(* Logix 5000 project; controller cal1632 1756-L62 rev 16.20; software revision 16.05; part 42 of 57 *)
(* tags used below, declared in another part *)
   FAULT : BOOL;
   HMI : BOOL;
   p01r09_pb_global_reset : BOOL;
   p02_real_from_hmi : hmi_real;
   p25_ai_amps : DINT;
   p25_ai_hz : DINT;
   p25_ai_rpm : REAL;
   p25_ai_speed : REAL;
   p25_ai_ts2_lc : REAL;
   p25_ao_selected_speed : REAL;
   p25_ao_torque : REAL;
   p25_ao_vfd : REAL;
   p25_control_word : INT;
   p25_di_brake : BOOL;
   p25_di_therm : BOOL;
   p25_di_ts2 : acs800_di_normal;
   p25_dint_to_hmi : DINT[16];
   p25_real_to_hmi : REAL[112];
   p25_status_word : INT;
   p25_ts2_gear_ratio : REAL;
   p25_ts2_roll_diameter_ft : REAL;
   p25_vfd_input_max : REAL;
   p25_vfd_input_min : REAL;
   p25_vfd_output_max : REAL;
   p25_vfd_output_min : REAL;
   p25r03_vfd_out_scaling : SYS_SCP;
   p25r04 : routine;
   p25r04_speed_to_vfd_ts2_scp : SYS_SPEED_TO_VFD;
   p25r04_timer_fault : TIMER[4];
   p25r04_timer_warning : TIMER[4];
   p25r05 : routine;
   p25r05_timer_fault : TIMER[4];
   p25r05_timer_warning : TIMER[4];
   p25r06 : routine;
   p25r06_ave_lc : REAL;
   p25r06_lc_ave_ctrl : CONTROL;
   p25r06_lc_buffer : REAL[20];
   p25r06_lc_ctrl : CONTROL;
   p25r06_sample_timer : TIMER;
   p25r06_timer_fault : TIMER[4];
   p25r06_timer_warning : TIMER[4];
   p25r06_unload : REAL;
   p25r07 : routine;
   p25r07_timer_fault : TIMER[4];
   p25r07_timer_warning : TIMER[4];
   p25r09_mode_jog : BOOL;
   p25r09_mode_run : BOOL;
   p25r09_mode_thread : BOOL;
   p25r11 : routine;
(* P25_Tension_Stand_2, continued *)

ROUTINE R04_Output   (* ladder *)
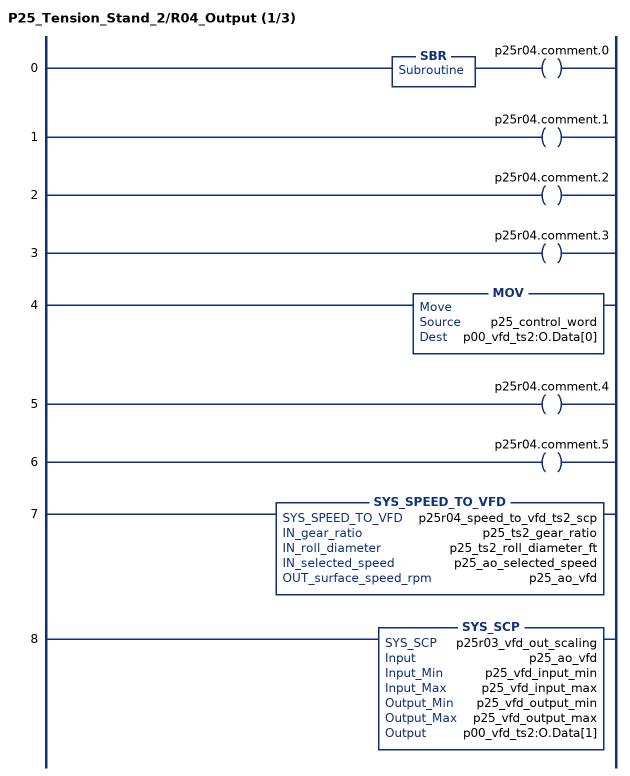
   0: SBR()OTE(p25r04.comment.0);
   1: OTE(p25r04.comment.1);
   2: OTE(p25r04.comment.2);
   3: OTE(p25r04.comment.3);
   4: MOV(p25_control_word,p00_vfd_ts2:O.Data[0]);
   5: OTE(p25r04.comment.4);
   6: OTE(p25r04.comment.5);
   7: SYS_SPEED_TO_VFD(p25r04_speed_to_vfd_ts2_scp,p25_ts2_gear_ratio,p25_ts2_roll_diameter_ft,p25_ao_selected_speed,p25_ao_vfd);
   8: SYS_SCP(p25r03_vfd_out_scaling,p25_ao_vfd,p25_vfd_input_min,p25_vfd_input_max,p25_vfd_output_min,p25_vfd_output_max,p00_vfd_ts2:O.Data[1]);
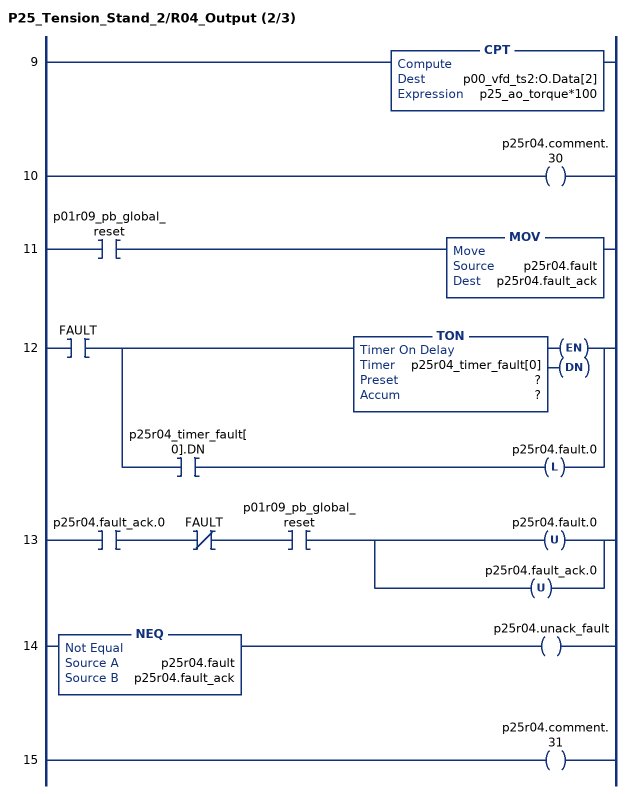
   9: CPT(p00_vfd_ts2:O.Data[2],p25_ao_torque*100);
   10: OTE(p25r04.comment.30);
   11: XIC(p01r09_pb_global_reset)MOV(p25r04.fault,p25r04.fault_ack);
   12: XIC(FAULT)[TON(p25r04_timer_fault[0],?,?) ,XIC(p25r04_timer_fault[0].DN) OTL(p25r04.fault.0) ];
   13: XIC(p25r04.fault_ack.0)XIO(FAULT)XIC(p01r09_pb_global_reset)[OTU(p25r04.fault.0) ,OTU(p25r04.fault_ack.0) ];
   14: NEQ(p25r04.fault,p25r04.fault_ack)OTE(p25r04.unack_fault);
   15: OTE(p25r04.comment.31);
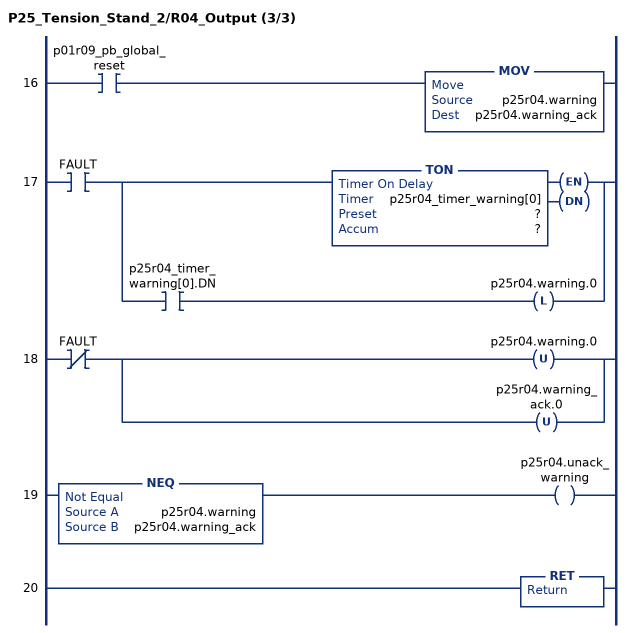
   16: XIC(p01r09_pb_global_reset)MOV(p25r04.warning,p25r04.warning_ack);
   17: XIC(FAULT)[TON(p25r04_timer_warning[0],?,?) ,XIC(p25r04_timer_warning[0].DN) OTL(p25r04.warning.0) ];
   18: XIO(FAULT)[OTU(p25r04.warning.0) ,OTU(p25r04.warning_ack.0) ];
   19: NEQ(p25r04.warning,p25r04.warning_ack)OTE(p25r04.unack_warning);
   20: RET();
END_ROUTINE

ROUTINE R05_Dint_to_HMI   (* ladder *)
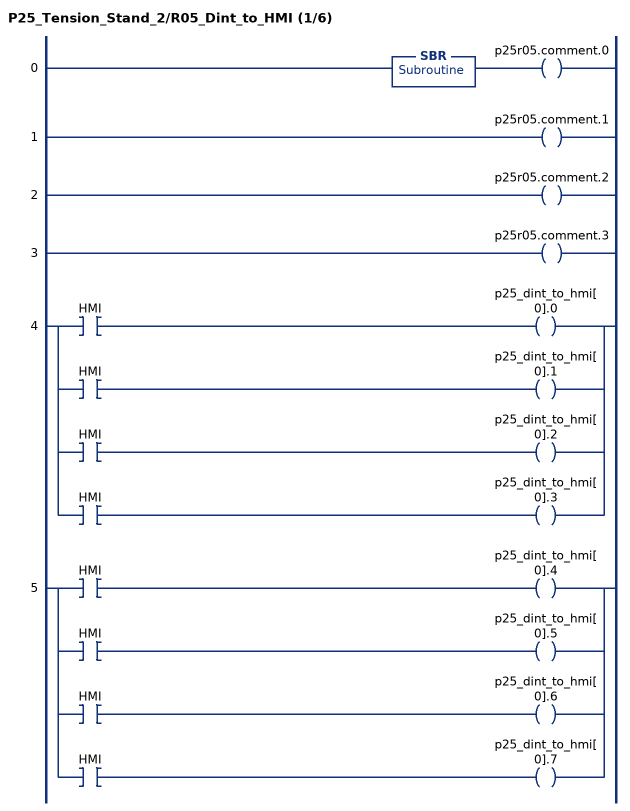
   0: SBR()OTE(p25r05.comment.0);
   1: OTE(p25r05.comment.1);
   2: OTE(p25r05.comment.2);
   3: OTE(p25r05.comment.3);
   4: [XIC(HMI) OTE(p25_dint_to_hmi[0].0) ,XIC(HMI) OTE(p25_dint_to_hmi[0].1) ,XIC(HMI) OTE(p25_dint_to_hmi[0].2) ,XIC(HMI) OTE(p25_dint_to_hmi[0].3) ];
   5: [XIC(HMI) OTE(p25_dint_to_hmi[0].4) ,XIC(HMI) OTE(p25_dint_to_hmi[0].5) ,XIC(HMI) OTE(p25_dint_to_hmi[0].6) ,XIC(HMI) OTE(p25_dint_to_hmi[0].7) ];
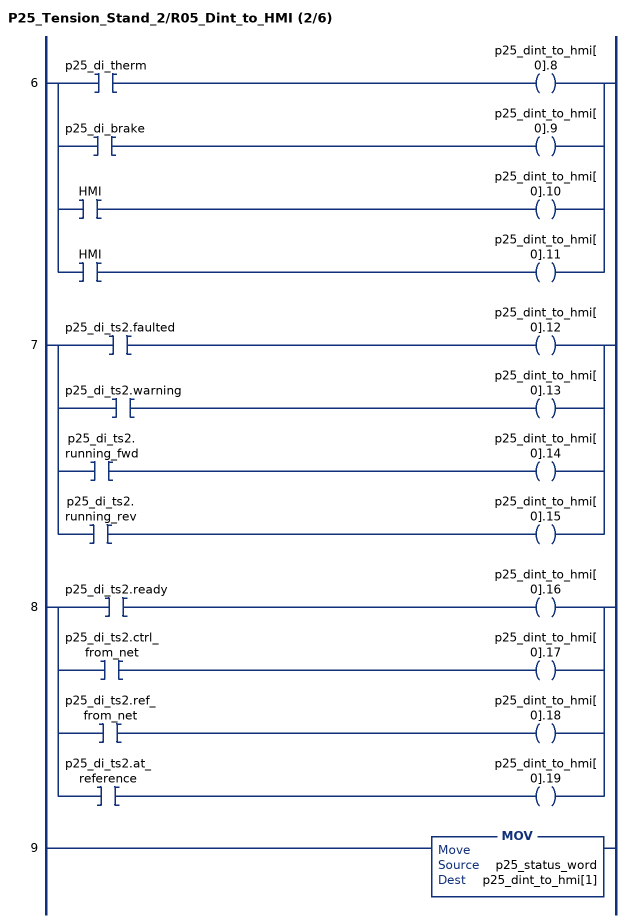
   6: [XIC(p25_di_therm) OTE(p25_dint_to_hmi[0].8) ,XIC(p25_di_brake) OTE(p25_dint_to_hmi[0].9) ,XIC(HMI) OTE(p25_dint_to_hmi[0].10) ,XIC(HMI) OTE(p25_dint_to_hmi[0].11) ];
   7: [XIC(p25_di_ts2.faulted) OTE(p25_dint_to_hmi[0].12) ,XIC(p25_di_ts2.warning) OTE(p25_dint_to_hmi[0].13) ,XIC(p25_di_ts2.running_fwd) OTE(p25_dint_to_hmi[0].14) ,XIC(p25_di_ts2.running_rev) OTE(p25_dint_to_hmi[0].15) ];
   8: [XIC(p25_di_ts2.ready) OTE(p25_dint_to_hmi[0].16) ,XIC(p25_di_ts2.ctrl_from_net) OTE(p25_dint_to_hmi[0].17) ,XIC(p25_di_ts2.ref_from_net) OTE(p25_dint_to_hmi[0].18) ,XIC(p25_di_ts2.at_reference) OTE(p25_dint_to_hmi[0].19) ];
   9: MOV(p25_status_word,p25_dint_to_hmi[1]);
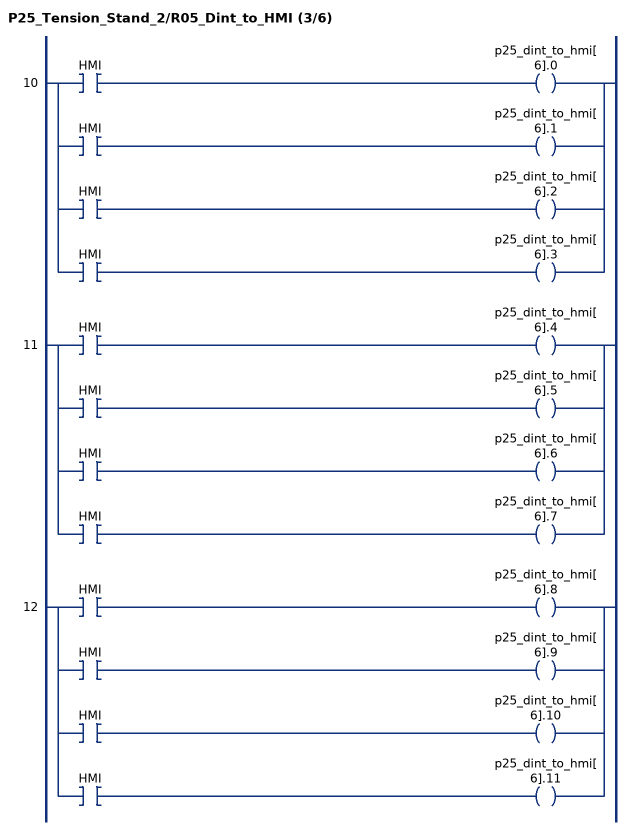
   10: [XIC(HMI) OTE(p25_dint_to_hmi[6].0) ,XIC(HMI) OTE(p25_dint_to_hmi[6].1) ,XIC(HMI) OTE(p25_dint_to_hmi[6].2) ,XIC(HMI) OTE(p25_dint_to_hmi[6].3) ];
   11: [XIC(HMI) OTE(p25_dint_to_hmi[6].4) ,XIC(HMI) OTE(p25_dint_to_hmi[6].5) ,XIC(HMI) OTE(p25_dint_to_hmi[6].6) ,XIC(HMI) OTE(p25_dint_to_hmi[6].7) ];
   12: [XIC(HMI) OTE(p25_dint_to_hmi[6].8) ,XIC(HMI) OTE(p25_dint_to_hmi[6].9) ,XIC(HMI) OTE(p25_dint_to_hmi[6].10) ,XIC(HMI) OTE(p25_dint_to_hmi[6].11) ];
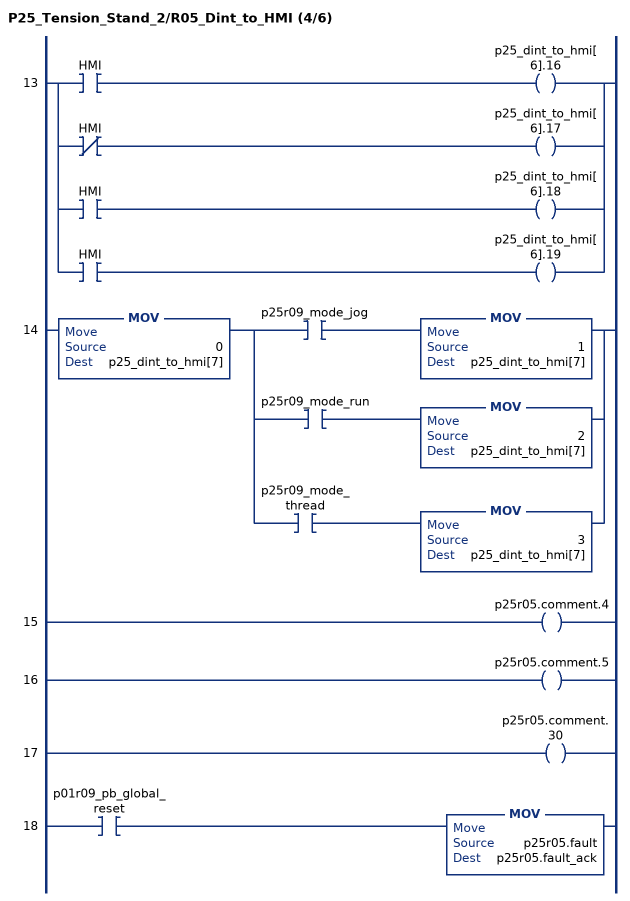
   13: [XIC(HMI) OTE(p25_dint_to_hmi[6].16) ,XIO(HMI) OTE(p25_dint_to_hmi[6].17) ,XIC(HMI) OTE(p25_dint_to_hmi[6].18) ,XIC(HMI) OTE(p25_dint_to_hmi[6].19) ];
   14: MOV(0,p25_dint_to_hmi[7])[XIC(p25r09_mode_jog) MOV(1,p25_dint_to_hmi[7]) ,XIC(p25r09_mode_run) MOV(2,p25_dint_to_hmi[7]) ,XIC(p25r09_mode_thread) MOV(3,p25_dint_to_hmi[7]) ];
   15: OTE(p25r05.comment.4);
   16: OTE(p25r05.comment.5);
   17: OTE(p25r05.comment.30);
   18: XIC(p01r09_pb_global_reset)MOV(p25r05.fault,p25r05.fault_ack);
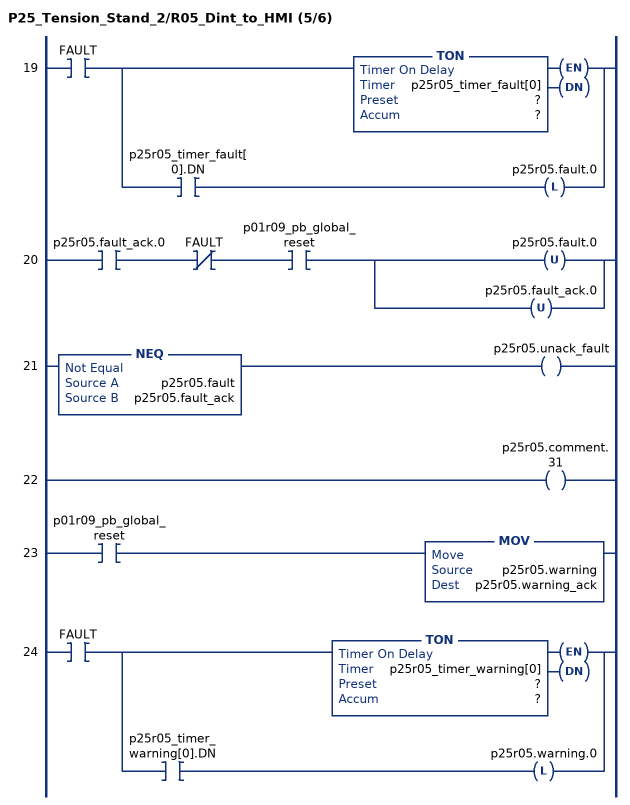
   19: XIC(FAULT)[TON(p25r05_timer_fault[0],?,?) ,XIC(p25r05_timer_fault[0].DN) OTL(p25r05.fault.0) ];
   20: XIC(p25r05.fault_ack.0)XIO(FAULT)XIC(p01r09_pb_global_reset)[OTU(p25r05.fault.0) ,OTU(p25r05.fault_ack.0) ];
   21: NEQ(p25r05.fault,p25r05.fault_ack)OTE(p25r05.unack_fault);
   22: OTE(p25r05.comment.31);
   23: XIC(p01r09_pb_global_reset)MOV(p25r05.warning,p25r05.warning_ack);
   24: XIC(FAULT)[TON(p25r05_timer_warning[0],?,?) ,XIC(p25r05_timer_warning[0].DN) OTL(p25r05.warning.0) ];
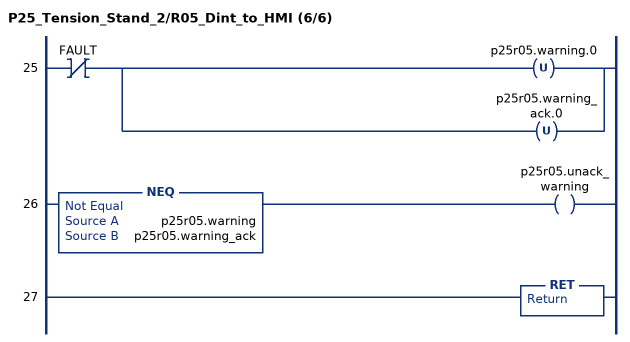
   25: XIO(FAULT)[OTU(p25r05.warning.0) ,OTU(p25r05.warning_ack.0) ];
   26: NEQ(p25r05.warning,p25r05.warning_ack)OTE(p25r05.unack_warning);
   27: RET();
END_ROUTINE

ROUTINE R06_Real_to_HMI   (* ladder *)
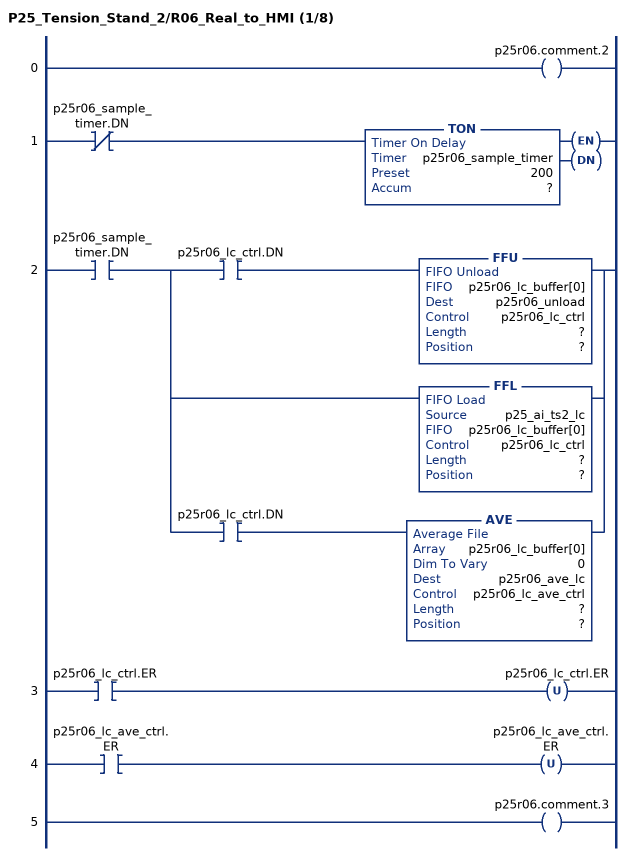
   0: OTE(p25r06.comment.2);
   1: XIO(p25r06_sample_timer.DN)TON(p25r06_sample_timer,?,?);
   2: XIC(p25r06_sample_timer.DN)[XIC(p25r06_lc_ctrl.DN) FFU(p25r06_lc_buffer[0],p25r06_unload,p25r06_lc_ctrl,?,?) ,FFL(p25_ai_ts2_lc,p25r06_lc_buffer[0],p25r06_lc_ctrl,?,?) ,XIC(p25r06_lc_ctrl.DN) AVE(p25r06_lc_buffer[0],0,p25r06_ave_lc,p25r06_lc_ave_ctrl,?,?) ];
   3: XIC(p25r06_lc_ctrl.ER)OTU(p25r06_lc_ctrl.ER);
   4: XIC(p25r06_lc_ave_ctrl.ER)OTU(p25r06_lc_ave_ctrl.ER);
   5: OTE(p25r06.comment.3);
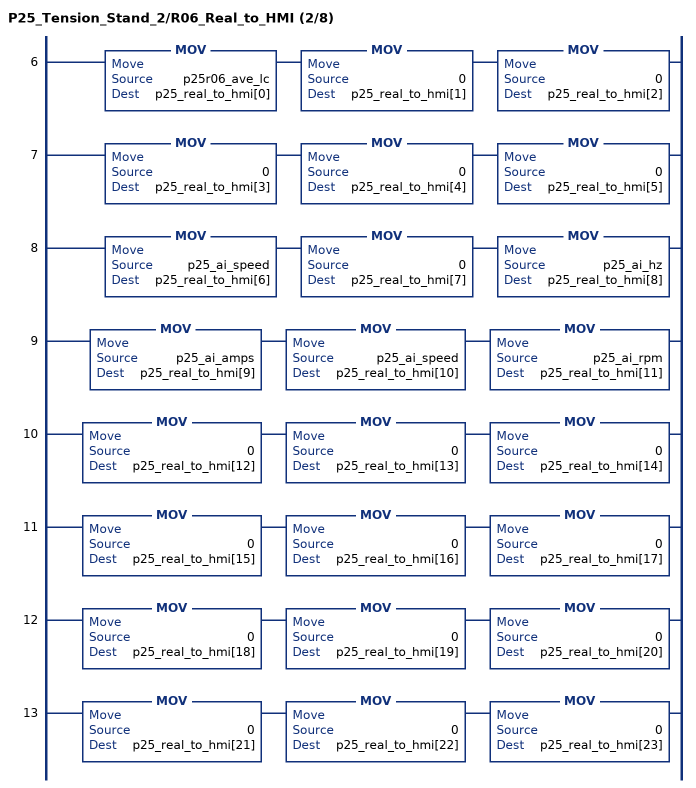
   6: MOV(p25r06_ave_lc,p25_real_to_hmi[0])MOV(0,p25_real_to_hmi[1])MOV(0,p25_real_to_hmi[2]);
   7: MOV(0,p25_real_to_hmi[3])MOV(0,p25_real_to_hmi[4])MOV(0,p25_real_to_hmi[5]);
   8: MOV(p25_ai_speed,p25_real_to_hmi[6])MOV(0,p25_real_to_hmi[7])MOV(p25_ai_hz,p25_real_to_hmi[8]);
   9: MOV(p25_ai_amps,p25_real_to_hmi[9])MOV(p25_ai_speed,p25_real_to_hmi[10])MOV(p25_ai_rpm,p25_real_to_hmi[11]);
   10: MOV(0,p25_real_to_hmi[12])MOV(0,p25_real_to_hmi[13])MOV(0,p25_real_to_hmi[14]);
   11: MOV(0,p25_real_to_hmi[15])MOV(0,p25_real_to_hmi[16])MOV(0,p25_real_to_hmi[17]);
   12: MOV(0,p25_real_to_hmi[18])MOV(0,p25_real_to_hmi[19])MOV(0,p25_real_to_hmi[20]);
   13: MOV(0,p25_real_to_hmi[21])MOV(0,p25_real_to_hmi[22])MOV(0,p25_real_to_hmi[23]);
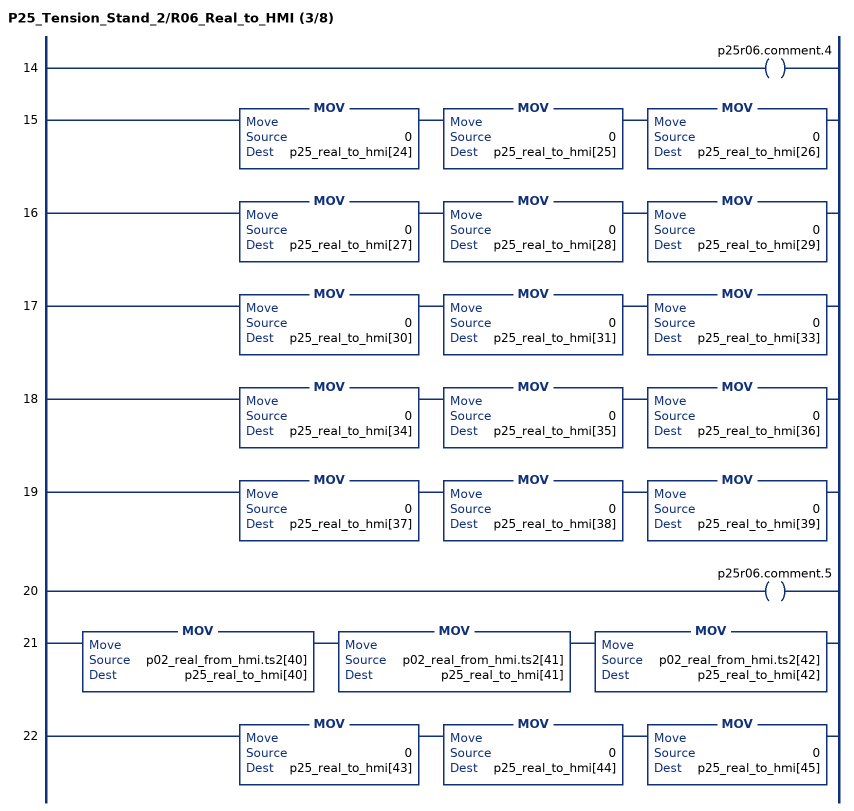
   14: OTE(p25r06.comment.4);
   15: MOV(0,p25_real_to_hmi[24])MOV(0,p25_real_to_hmi[25])MOV(0,p25_real_to_hmi[26]);
   16: MOV(0,p25_real_to_hmi[27])MOV(0,p25_real_to_hmi[28])MOV(0,p25_real_to_hmi[29]);
   17: MOV(0,p25_real_to_hmi[30])MOV(0,p25_real_to_hmi[31])MOV(0,p25_real_to_hmi[33]);
   18: MOV(0,p25_real_to_hmi[34])MOV(0,p25_real_to_hmi[35])MOV(0,p25_real_to_hmi[36]);
   19: MOV(0,p25_real_to_hmi[37])MOV(0,p25_real_to_hmi[38])MOV(0,p25_real_to_hmi[39]);
   20: OTE(p25r06.comment.5);
   21: MOV(p02_real_from_hmi.ts2[40],p25_real_to_hmi[40])MOV(p02_real_from_hmi.ts2[41],p25_real_to_hmi[41])MOV(p02_real_from_hmi.ts2[42],p25_real_to_hmi[42]);
   22: MOV(0,p25_real_to_hmi[43])MOV(0,p25_real_to_hmi[44])MOV(0,p25_real_to_hmi[45]);
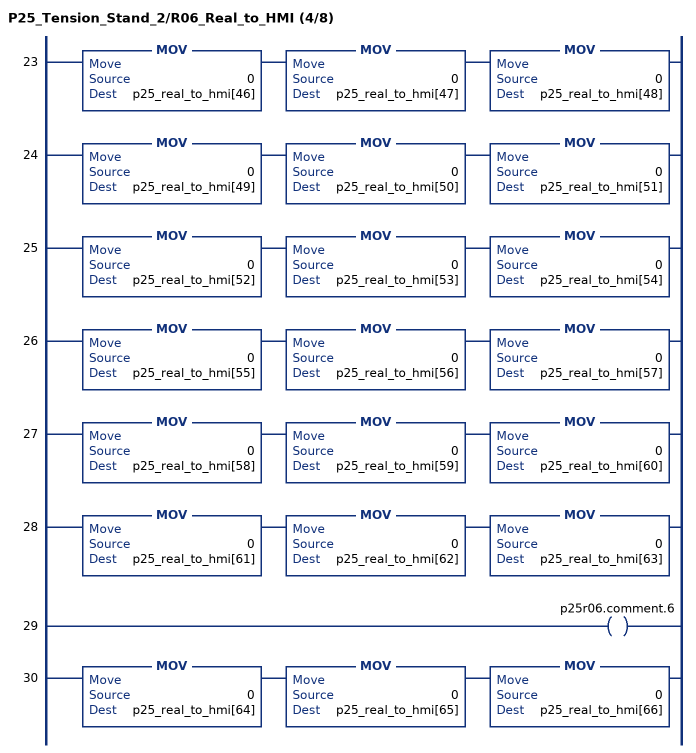
   23: MOV(0,p25_real_to_hmi[46])MOV(0,p25_real_to_hmi[47])MOV(0,p25_real_to_hmi[48]);
   24: MOV(0,p25_real_to_hmi[49])MOV(0,p25_real_to_hmi[50])MOV(0,p25_real_to_hmi[51]);
   25: MOV(0,p25_real_to_hmi[52])MOV(0,p25_real_to_hmi[53])MOV(0,p25_real_to_hmi[54]);
   26: MOV(0,p25_real_to_hmi[55])MOV(0,p25_real_to_hmi[56])MOV(0,p25_real_to_hmi[57]);
   27: MOV(0,p25_real_to_hmi[58])MOV(0,p25_real_to_hmi[59])MOV(0,p25_real_to_hmi[60]);
   28: MOV(0,p25_real_to_hmi[61])MOV(0,p25_real_to_hmi[62])MOV(0,p25_real_to_hmi[63]);
   29: OTE(p25r06.comment.6);
   30: MOV(0,p25_real_to_hmi[64])MOV(0,p25_real_to_hmi[65])MOV(0,p25_real_to_hmi[66]);
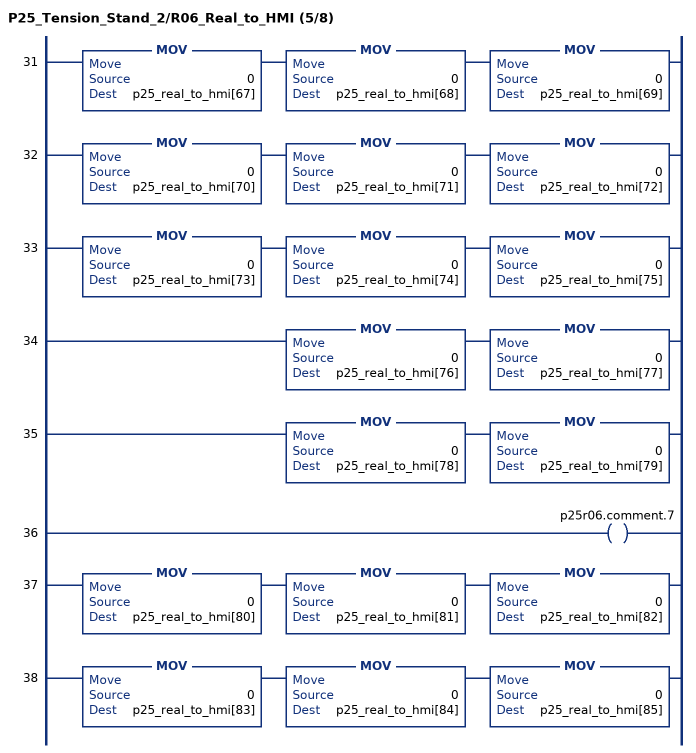
   31: MOV(0,p25_real_to_hmi[67])MOV(0,p25_real_to_hmi[68])MOV(0,p25_real_to_hmi[69]);
   32: MOV(0,p25_real_to_hmi[70])MOV(0,p25_real_to_hmi[71])MOV(0,p25_real_to_hmi[72]);
   33: MOV(0,p25_real_to_hmi[73])MOV(0,p25_real_to_hmi[74])MOV(0,p25_real_to_hmi[75]);
   34: MOV(0,p25_real_to_hmi[76])MOV(0,p25_real_to_hmi[77]);
   35: MOV(0,p25_real_to_hmi[78])MOV(0,p25_real_to_hmi[79]);
   36: OTE(p25r06.comment.7);
   37: MOV(0,p25_real_to_hmi[80])MOV(0,p25_real_to_hmi[81])MOV(0,p25_real_to_hmi[82]);
   38: MOV(0,p25_real_to_hmi[83])MOV(0,p25_real_to_hmi[84])MOV(0,p25_real_to_hmi[85]);
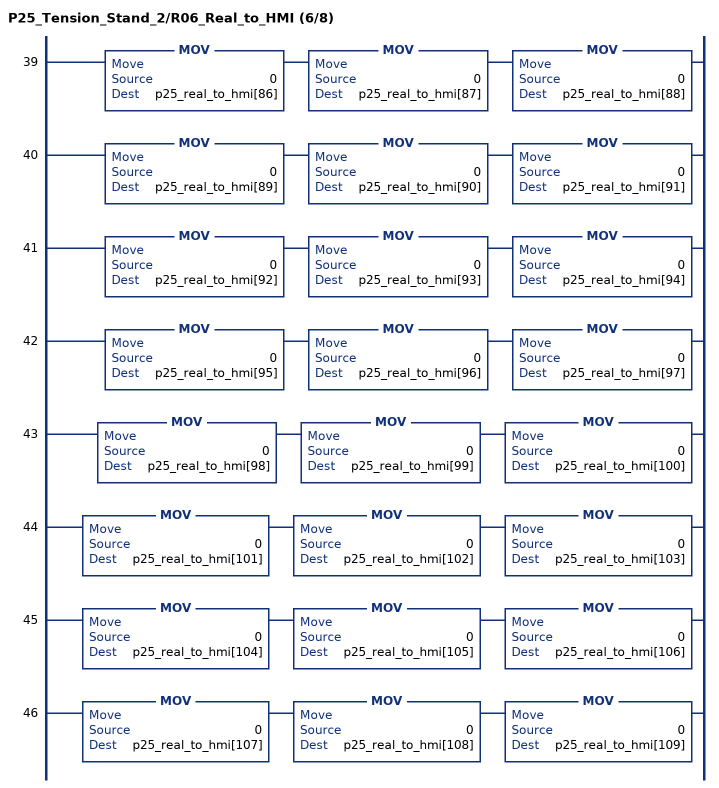
   39: MOV(0,p25_real_to_hmi[86])MOV(0,p25_real_to_hmi[87])MOV(0,p25_real_to_hmi[88]);
   40: MOV(0,p25_real_to_hmi[89])MOV(0,p25_real_to_hmi[90])MOV(0,p25_real_to_hmi[91]);
   41: MOV(0,p25_real_to_hmi[92])MOV(0,p25_real_to_hmi[93])MOV(0,p25_real_to_hmi[94]);
   42: MOV(0,p25_real_to_hmi[95])MOV(0,p25_real_to_hmi[96])MOV(0,p25_real_to_hmi[97]);
   43: MOV(0,p25_real_to_hmi[98])MOV(0,p25_real_to_hmi[99])MOV(0,p25_real_to_hmi[100]);
   44: MOV(0,p25_real_to_hmi[101])MOV(0,p25_real_to_hmi[102])MOV(0,p25_real_to_hmi[103]);
   45: MOV(0,p25_real_to_hmi[104])MOV(0,p25_real_to_hmi[105])MOV(0,p25_real_to_hmi[106]);
   46: MOV(0,p25_real_to_hmi[107])MOV(0,p25_real_to_hmi[108])MOV(0,p25_real_to_hmi[109]);
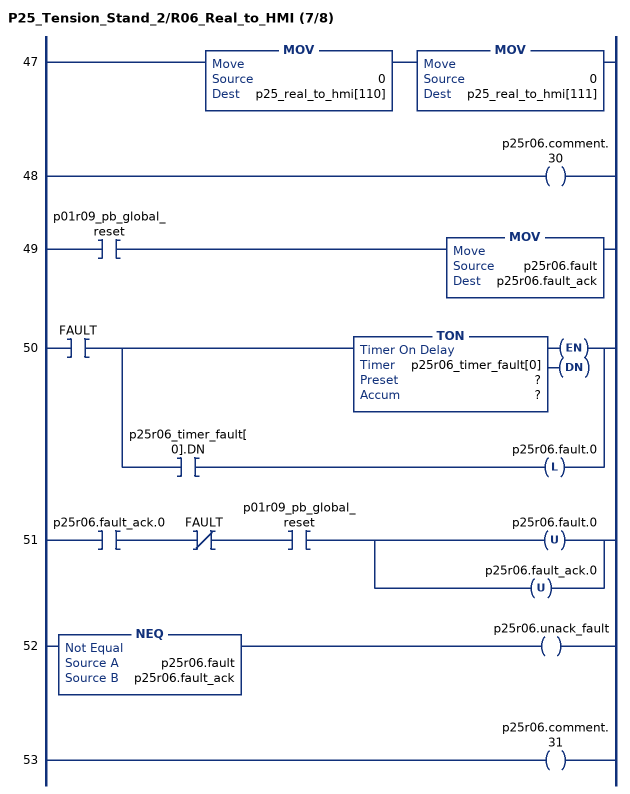
   47: MOV(0,p25_real_to_hmi[110])MOV(0,p25_real_to_hmi[111]);
   48: OTE(p25r06.comment.30);
   49: XIC(p01r09_pb_global_reset)MOV(p25r06.fault,p25r06.fault_ack);
   50: XIC(FAULT)[TON(p25r06_timer_fault[0],?,?) ,XIC(p25r06_timer_fault[0].DN) OTL(p25r06.fault.0) ];
   51: XIC(p25r06.fault_ack.0)XIO(FAULT)XIC(p01r09_pb_global_reset)[OTU(p25r06.fault.0) ,OTU(p25r06.fault_ack.0) ];
   52: NEQ(p25r06.fault,p25r06.fault_ack)OTE(p25r06.unack_fault);
   53: OTE(p25r06.comment.31);
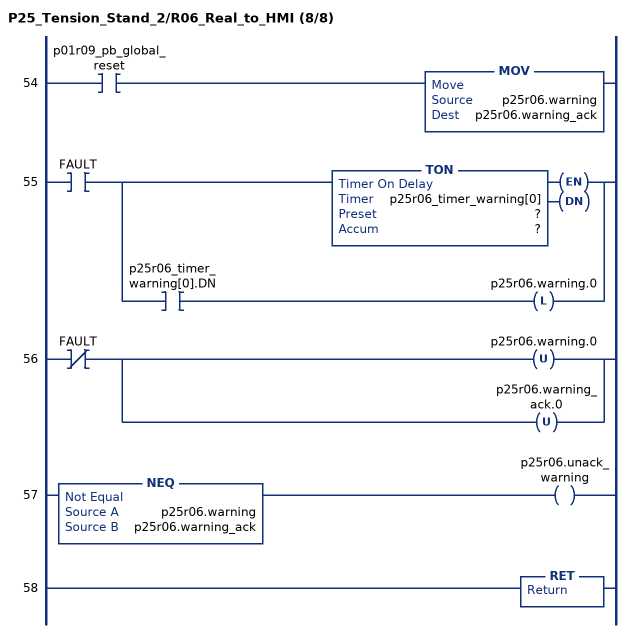
   54: XIC(p01r09_pb_global_reset)MOV(p25r06.warning,p25r06.warning_ack);
   55: XIC(FAULT)[TON(p25r06_timer_warning[0],?,?) ,XIC(p25r06_timer_warning[0].DN) OTL(p25r06.warning.0) ];
   56: XIO(FAULT)[OTU(p25r06.warning.0) ,OTU(p25r06.warning_ack.0) ];
   57: NEQ(p25r06.warning,p25r06.warning_ack)OTE(p25r06.unack_warning);
   58: RET();
END_ROUTINE

ROUTINE R07_Alarms   (* ladder *)
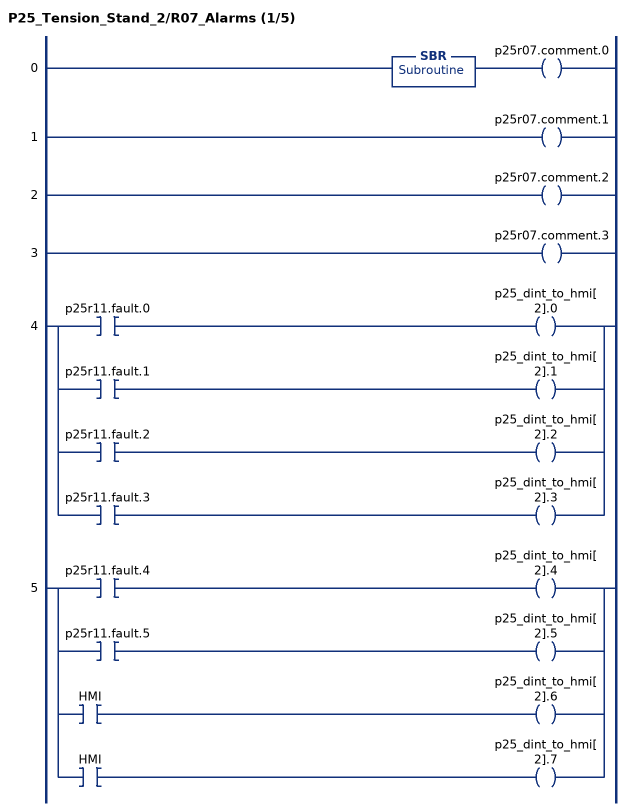
   0: SBR()OTE(p25r07.comment.0);
   1: OTE(p25r07.comment.1);
   2: OTE(p25r07.comment.2);
   3: OTE(p25r07.comment.3);
   4: [XIC(p25r11.fault.0) OTE(p25_dint_to_hmi[2].0) ,XIC(p25r11.fault.1) OTE(p25_dint_to_hmi[2].1) ,XIC(p25r11.fault.2) OTE(p25_dint_to_hmi[2].2) ,XIC(p25r11.fault.3) OTE(p25_dint_to_hmi[2].3) ];
   5: [XIC(p25r11.fault.4) OTE(p25_dint_to_hmi[2].4) ,XIC(p25r11.fault.5) OTE(p25_dint_to_hmi[2].5) ,XIC(HMI) OTE(p25_dint_to_hmi[2].6) ,XIC(HMI) OTE(p25_dint_to_hmi[2].7) ];
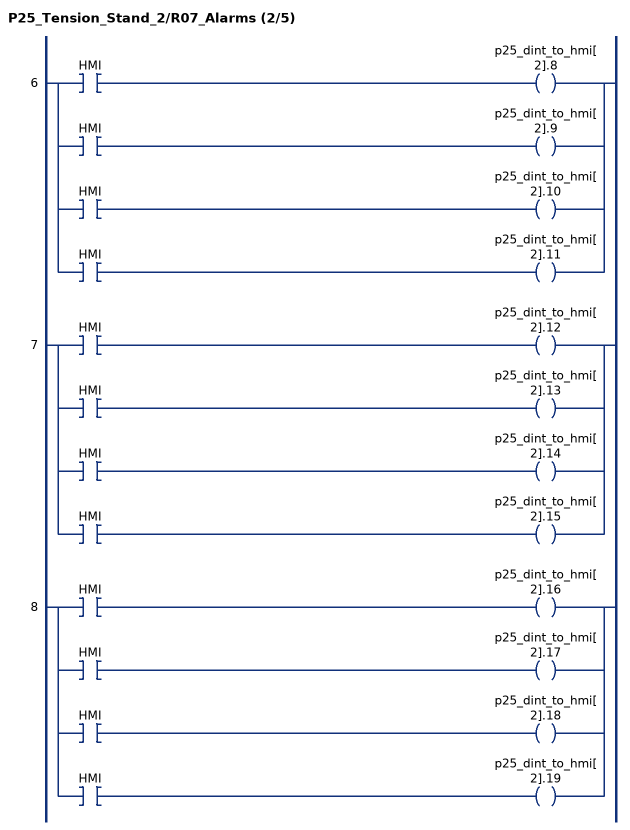
   6: [XIC(HMI) OTE(p25_dint_to_hmi[2].8) ,XIC(HMI) OTE(p25_dint_to_hmi[2].9) ,XIC(HMI) OTE(p25_dint_to_hmi[2].10) ,XIC(HMI) OTE(p25_dint_to_hmi[2].11) ];
   7: [XIC(HMI) OTE(p25_dint_to_hmi[2].12) ,XIC(HMI) OTE(p25_dint_to_hmi[2].13) ,XIC(HMI) OTE(p25_dint_to_hmi[2].14) ,XIC(HMI) OTE(p25_dint_to_hmi[2].15) ];
   8: [XIC(HMI) OTE(p25_dint_to_hmi[2].16) ,XIC(HMI) OTE(p25_dint_to_hmi[2].17) ,XIC(HMI) OTE(p25_dint_to_hmi[2].18) ,XIC(HMI) OTE(p25_dint_to_hmi[2].19) ];
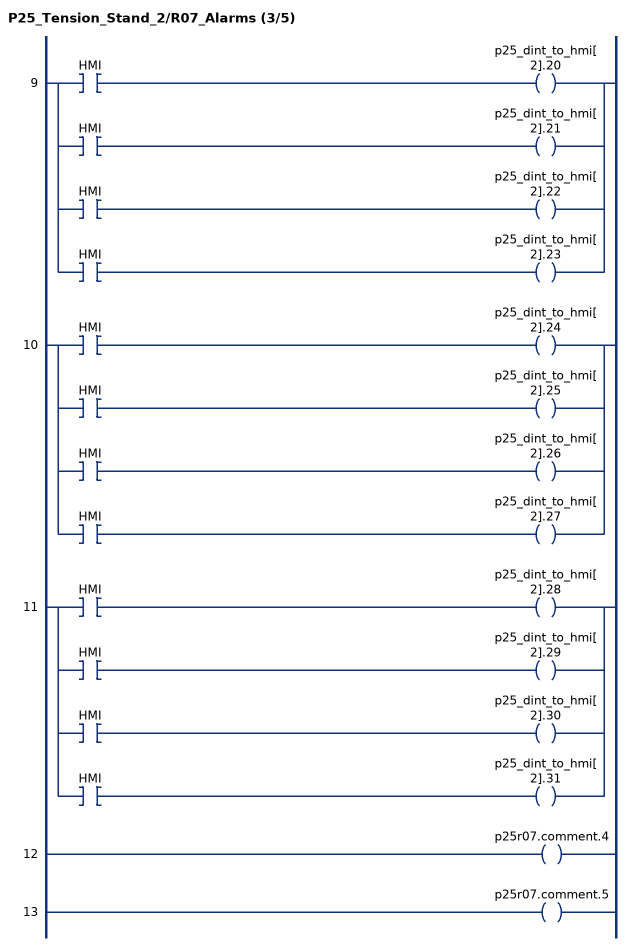
   9: [XIC(HMI) OTE(p25_dint_to_hmi[2].20) ,XIC(HMI) OTE(p25_dint_to_hmi[2].21) ,XIC(HMI) OTE(p25_dint_to_hmi[2].22) ,XIC(HMI) OTE(p25_dint_to_hmi[2].23) ];
   10: [XIC(HMI) OTE(p25_dint_to_hmi[2].24) ,XIC(HMI) OTE(p25_dint_to_hmi[2].25) ,XIC(HMI) OTE(p25_dint_to_hmi[2].26) ,XIC(HMI) OTE(p25_dint_to_hmi[2].27) ];
   11: [XIC(HMI) OTE(p25_dint_to_hmi[2].28) ,XIC(HMI) OTE(p25_dint_to_hmi[2].29) ,XIC(HMI) OTE(p25_dint_to_hmi[2].30) ,XIC(HMI) OTE(p25_dint_to_hmi[2].31) ];
   12: OTE(p25r07.comment.4);
   13: OTE(p25r07.comment.5);
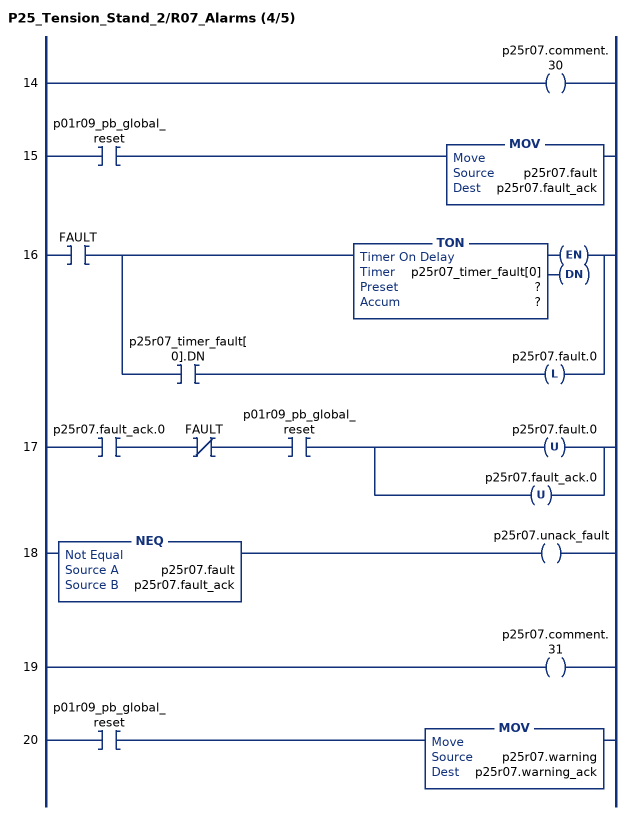
   14: OTE(p25r07.comment.30);
   15: XIC(p01r09_pb_global_reset)MOV(p25r07.fault,p25r07.fault_ack);
   16: XIC(FAULT)[TON(p25r07_timer_fault[0],?,?) ,XIC(p25r07_timer_fault[0].DN) OTL(p25r07.fault.0) ];
   17: XIC(p25r07.fault_ack.0)XIO(FAULT)XIC(p01r09_pb_global_reset)[OTU(p25r07.fault.0) ,OTU(p25r07.fault_ack.0) ];
   18: NEQ(p25r07.fault,p25r07.fault_ack)OTE(p25r07.unack_fault);
   19: OTE(p25r07.comment.31);
   20: XIC(p01r09_pb_global_reset)MOV(p25r07.warning,p25r07.warning_ack);
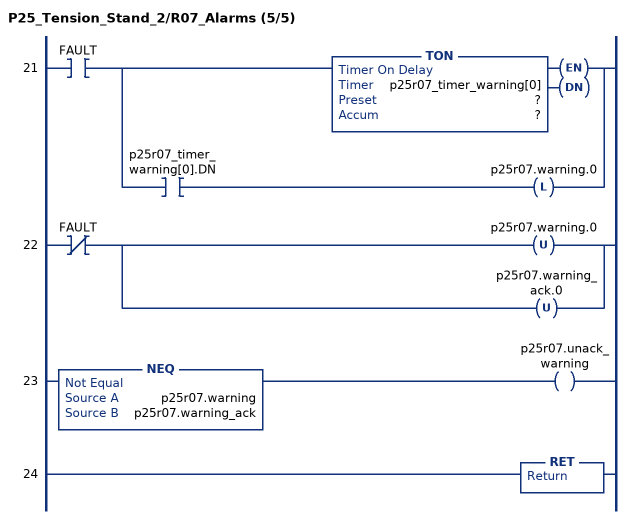
   21: XIC(FAULT)[TON(p25r07_timer_warning[0],?,?) ,XIC(p25r07_timer_warning[0].DN) OTL(p25r07.warning.0) ];
   22: XIO(FAULT)[OTU(p25r07.warning.0) ,OTU(p25r07.warning_ack.0) ];
   23: NEQ(p25r07.warning,p25r07.warning_ack)OTE(p25r07.unack_warning);
   24: RET();
END_ROUTINE
